TYPE DUT_stSPAlarm :
STRUCT
	Error : BOOL;
	ErrorID : DINT;
END_STRUCT
END_TYPE

(* stored: Version 1.1.0.1, ProductVersion 3.1.4024.15
   DUT DUT_stSPAlarm: Id {dcd8db16-76ff-415f-b45a-e972c4d6f9c3} *)
